FUNCTION_BLOCK Test_TStreamAdd_Read_PVOID EXTENDS T_UnitTestBase
VAR
    Stream  : T_Stream(StreamLength := 2);
    ArgType : E_ArgTypeId := E_ArgTypeId.Type_PVOID;
    Bob     : INT;
END_VAR

Stream.Init(2);

// add a pointer...
Stream.SetNextArgTypeId(ArgType);
Stream.Add_PVOID(ADR(Bob));

Stream.SetReadPosition(0);

// check next arg type is correct...
Assertion.AssertEquals_INT(Expected     := ArgType,
                           Actual       := Stream.GetNextArgTypeId(),
                           VariableName := 'Stream.GetNextArgTypeId()');

// check next value...	
Assertion.AssertEquals_PVOID(Expected     := ADR(Bob),
                             Actual       := Stream.Read_PVOID(),
                             VariableName := 'Stream.Read_PVOID()');

// check we are at the end of the stream..							
Assertion.AssertEquals_UDINT(Expected     := Stream.StreamLength,
                             Actual       := Stream.ReadPosition,
                             VariableName := 'Stream.ReadPosition');

TestFinished();

END_FUNCTION_BLOCK

(* stored: Version 1.1.0.1, ProductVersion 3.1.4024.11
   POU Test_TStreamAdd_Read_PVOID: Id {f56765ee-e2ea-44a1-a75c-6f5827ff678e}, SpecialFunc None *)
